# EPICS autosave request: roles/install_ioc/tasks/device_types/mrftiming/files/auto_settings.req
file "vme-evr-230rf.req",       P=$(P),  R=$(R)
